TYPE ST_MasterCoupling :
STRUCT
	iMasterAxis		:	UINT	:=1;		//Must be initialised to 1 as no 0 index on arrays
	eLimitType		:	eLimitCoupling;
END_STRUCT
END_TYPE

(* stored: Version 1.1.0.1, ProductVersion 3.1.4022.12
   DUT ST_MasterCoupling: Id {91d98661-f043-491d-b94f-39405d5fb838} *)
